FUNCTION_BLOCK FB_ElementB IMPLEMENTS I_VisitibleElement
VAR_INPUT
END_VAR
VAR_OUTPUT
END_VAR
VAR
END_VAR

METHOD accept
VAR_INPUT
	in_ipVisitor	: I_Visitor;
END_VAR
in_ipVisitor.VisitElementB(in_fbElementB:= THIS^);
END_METHOD

END_FUNCTION_BLOCK

(* stored: Version 1.1.0.1
   POU FB_ElementB: Id {599073bd-6358-422a-8d7f-a088b040e299}, SpecialFunc None
   Method accept: Id {0b434423-c90c-4089-b877-d5136789fa73} *)
